# EPICS autosave request: iocBoot/ioc13XRM/auto_positions.req
file "CARS_motor_positions.req",      P=13XRM:, M=m1
file "CARS_motor_positions.req",      P=13XRM:, M=m2
file "CARS_motor_positions.req",      P=13XRM:, M=m3
file "CARS_motor_positions.req",      P=13XRM:, M=m4
file "CARS_motor_positions.req",      P=13XRM:, M=m5
file "CARS_motor_positions.req",      P=13XRM:, M=m6
file "CARS_motor_positions.req",      P=13XRM:, M=m7
file "CARS_motor_positions.req",      P=13XRM:, M=m8
# file "CARS_motor_positions.req",      P=13XRM:, M=m9
# file "CARS_motor_positions.req",      P=13XRM:, M=m10
# file "CARS_motor_positions.req",      P=13XRM:, M=m11
# file "CARS_motor_positions.req",      P=13XRM:, M=m12
